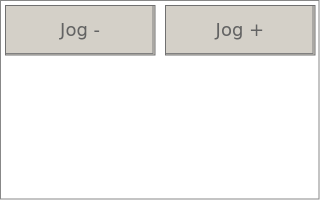
VISUALIZATION SingleAxisJogStandardFlast_1  // 320x200
VAR_IN_OUT
	btnJogPositive	: BOOL;
	btnJogNegative	: BOOL;
END_VAR
    Button (5,5 150x50), "Jog -"
        tap btnJogNegative
    Button (165,5 150x50), "Jog +"
        tap btnJogPositive
END_VISUALIZATION

(* stored: Version 1.1.0.1, ProductVersion 3.1.4024.12
   Visu SingleAxisJogStandardFlast_1: Id {56259215-3a01-47d6-979d-ad88df7bea20} *)
